(* Logix 5000 project; controller AplicacionAFEbancoDePruebas vendor 1 type 14 code 149 rev 33.12; software revision 33.01 *)

TASK MainTask (continuous, watchdog 500 ms) : MainProgram

MODULES
   Local : vendor 1 type 14 code 149 (Compact 0, rev 33.12)
      Discrete_IO : Embedded (Compact 1, rev 3.1, Output RPI 20 ms)
      PLC : 1769-L32E Ethernet Port (Ethernet 192.168.2.131, rev 20.1)
         PLC_Controller : vendor 1 type 14 code 77 (CompactLogixL32EController 0, rev 20.1, $6f3b489b$ RPI 20 ms, $fb73b292$ RPI 20 ms, $0a2ffb0d$ RPI 20 ms)
      VSD_AFE : vendor 1 type 143 code 8336 (Ethernet 192.168.2.50, rev 6.5, Output RPI 20 ms)
           VSD_AFE:O.LogicCommand_Stop   // Comando de Parada
           VSD_AFE:O.LogicCommand_Start   // Comando de Arranque
          : vendor 1 type 143 code 161 (RhinoBP 10, rev 1.1)
          : vendor 1 type 143 code 416 (RhinoBP 5, rev 1.8)
          : vendor 1 type 143 code 675 (RhinoBP 13, rev 1.1)
          : vendor 1 type 143 code 416 (RhinoBP 4, rev 1.8)
          : vendor 1 type 143 code 4770 (RhinoBP 12, rev 1.1)
          : vendor 1 type 143 code 2724 (RhinoBP 14, rev 1.1)
END_MODULES

TYPE Dinagrama :   // Estructura para el dinagrama
STRUCT
   vPotencia : REAL[500];   // captura del vector de potencia
   vCarga : REAL[500];   // captura del vector de carga
   vPosicion : REAL[500];   // captura del vector posicion
   vProximetro : DINT[500];   // captura del vector del proximetro
   NumeroMuestras : INT;
   enabled : BOOL;
   captura : BOOL;   // Flag que indica la captura del sistema
   resetVector : BOOL;   // Flag para darle Reset al vector de posición y carga
   vEmptyREAL : REAL[500];
   vEmptyINT : DINT[500];
   tMuestreo : REAL;   // Tiempo de Muestreo de captura
END_STRUCT
END_TYPE

TYPE LSW :   // Drive - Logic Status Word
STRUCT
   Faulted : BOOL;
   Warning : BOOL;
   RunForward : BOOL;
   RunReverse : BOOL;
   Ready : BOOL;
   RemoteRef : BOOL;
   RemoteCrtl : BOOL;
   AtSpeed : BOOL;
END_STRUCT
END_TYPE

TYPE SWC :
STRUCT
   Dinagrama : Dinagrama;
   VSD : VSD;
   entradasDigitales : INT;   // Entradas Digitales
   salidasDigitales : INT;   // Salidas Digitales
   entradasAnalogas : REAL[4];   // Entradas Analogas del PLC
   salidasAnalogas : REAL[4];
END_STRUCT
END_TYPE

TYPE VSD :   // VSD
STRUCT
   VSD_O : AB:PowerFlex755T_E_31635488:O:0;
   VSD_I : AB:PowerFlex755T_E_2B0A69C5:I:0;
END_STRUCT
END_TYPE

VAR_GLOBAL   (* controller tags *)
   SRP_Displacement_Actual : REAL := 22.99865;   // Variable de Simulacion PLC DC de Desplazamiento
   SRP_Load_Actual : REAL := 11.655421;   // Variable de simulacion PLC DC de Carga
   SRP_SimActualStroke : DINT;   // Variable Simulación de PLC Variador DC
   SWC : SWC := (Dinagrama.vCarga[0] := 9.6614, Dinagrama.vCarga[1] := 9.7812, Dinagrama.vCarga[2] := 9.711983, Dinagrama.vCarga[3] := 9.725293, Dinagrama.vCarga[4] := 9.842433, Dinagrama.vCarga[5] := 9.749254, Dinagrama.vCarga[6] := 9.69601, Dinagrama.vCarga[7] := 9.7306185, Dinagrama.vCarga[8] := 9.586858, Dinagrama.vCarga[9] := 9.751916, Dinagrama.vCarga[10] := 10.223133, Dinagrama.vCarga[11] := 10.473384, Dinagrama.vCarga[12] := 10.633119, Dinagrama.vCarga[13] := 10.856748, Dinagrama.vCarga[14] := 10.928628, Dinagrama.vCarga[15] := 11.109661, Dinagrama.vCarga[16] := 11.419147, Dinagrama.vCarga[17] := 11.515653, Dinagrama.vCarga[18] := 11.572558, Dinagrama.vCarga[19] := 11.751262, Dinagrama.vCarga[20] := 11.839782, Dinagrama.vCarga[21] := 11.974224, Dinagrama.vCarga[22] := 11.854091, Dinagrama.vCarga[23] := 11.607167, Dinagrama.vCarga[24] := 11.27239, Dinagrama.vCarga[25] := 11.069394, Dinagrama.vCarga[26] := 10.880708, Dinagrama.vCarga[27] := 10.662403, Dinagrama.vCarga[28] := 10.492021, Dinagrama.vCarga[29] := 10.321636, Dinagrama.vCarga[30] := 10.193849, Dinagrama.vCarga[31] := 10.018141, Dinagrama.vCarga[32] := 9.842432, Dinagrama.vCarga[33] := 9.682698, Dinagrama.vCarga[34] := 9.586857, Dinagrama.vCarga[35] := 9.706658, Dinagrama.vCarga[36] := 9.938273, Dinagrama.vCarga[37] := 10.113981, Dinagrama.vCarga[38] := 10.241769, Dinagrama.vCarga[39] := 10.321636, Dinagrama.vCarga[40] := 10.409491, Dinagrama.vCarga[41] := 10.409491, Dinagrama.vCarga[42] := 10.457411, Dinagrama.vCarga[43] := 10.534616, Dinagrama.vCarga[44] := 10.481371, Dinagrama.vCarga[45] := 10.555914, Dinagrama.vCarga[46] := 10.705, Dinagrama.vCarga[47] := 10.603834, Dinagrama.vCarga[48] := 10.316312, Dinagrama.vCarga[49] := 10.060737, Dinagrama.vCarga[50] := 9.970221, Dinagrama.vCarga[51] := 9.850419, Dinagrama.vCarga[52] := 9.608155, Dinagrama.vCarga[53] := 9.405825, Dinagrama.vCarga[54] := 9.389851, Dinagrama.vCarga[55] := 9.34193, Dinagrama.vCarga[56] := 9.131613, Dinagrama.vCarga[57] := 9.049084, Dinagrama.vCarga[58] := 9.08103, Dinagrama.vCarga[59] := 8.9266205,
        Dinagrama.vCarga[60] := 8.873376, Dinagrama.vCarga[61] := 9.155573, Dinagrama.vCarga[62] := 9.427122, Dinagrama.vCarga[63] := 9.549585, Dinagrama.vCarga[64] := 9.682697, Dinagrama.vCarga[65] := 9.906326, Dinagrama.vCarga[66] := 10.002167, Dinagrama.vCarga[67] := 9.980869, Dinagrama.vCarga[68] := 9.986194, Dinagrama.vCarga[69] := 9.980869, Dinagrama.vCarga[70] := 10.0208025, Dinagrama.vCarga[71] := 9.994181, Dinagrama.vCarga[72] := 10.098008, Dinagrama.vCarga[73] := 10.193849, Dinagrama.vCarga[74] := 9.938273, Dinagrama.vCarga[75] := 9.618804, Dinagrama.vCarga[76] := 9.538937, Dinagrama.vCarga[77] := 9.55491, Dinagrama.vCarga[78] := 9.331282, Dinagrama.vCarga[79] := 9.171547, Dinagrama.vCarga[80] := 9.347255, Dinagrama.vCarga[81] := 9.315308, Dinagrama.vCarga[82] := 9.123626, Dinagrama.vCarga[83] := 9.18752, Dinagrama.vCarga[84] := 9.331282, Dinagrama.vCarga[85] := 9.182196, Dinagrama.vCarga[86] := 9.166222, Dinagrama.vCarga[87] := 9.400499, Dinagrama.vCarga[88] := 9.693347, Dinagrama.vCarga[89] := 9.688023, Dinagrama.vCarga[90] := 9.746592, Dinagrama.vCarga[91] := 9.842432, Dinagrama.vCarga[92] := 9.885028, Dinagrama.vCarga[93] := 9.714644, Dinagrama.vCarga[94] := 9.634777, Dinagrama.vCarga[95] := 9.656075, Dinagrama.vCarga[96] := 9.496341, Dinagrama.vCarga[97] := 9.272713, Dinagrama.vCarga[98] := 9.128951, Dinagrama.vCarga[99] := 8.910647, Dinagrama.vCarga[100] := 8.434105, Dinagrama.vCarga[101] := 8.02412, Dinagrama.vCarga[102] := 7.936266, Dinagrama.vCarga[103] := 7.851074, Dinagrama.vCarga[104] := 7.5129685, Dinagrama.vCarga[105] := 7.302651, Dinagrama.vCarga[106] := 7.281353, Dinagrama.vCarga[107] := 7.238757, Dinagrama.vCarga[108] := 6.993831, Dinagrama.vCarga[109] := 6.706309, Dinagrama.vCarga[110] := 6.6796865, Dinagrama.vCarga[111] := 6.903315, Dinagrama.vCarga[112] := 7.1056457, Dinagrama.vCarga[113] := 7.3771944, Dinagrama.vCarga[114] := 7.773869, Dinagrama.vCarga[115] := 7.91763, Dinagrama.vCarga[116] := 7.909643, Dinagrama.vCarga[117] := 8.077365, Dinagrama.vCarga[118] := 8.300993, Dinagrama.vCarga[119] := 8.340926,
        Dinagrama.vCarga[120] := 8.460728, Dinagrama.vCarga[121] := 8.70033, Dinagrama.vCarga[122] := 8.79617, Dinagrama.vCarga[123] := 8.788184, Dinagrama.vCarga[124] := 8.77221, Dinagrama.vCarga[125] := 8.588515, Dinagrama.vCarga[126] := 8.38086, Dinagrama.vCarga[127] := 8.412807, Dinagrama.vCarga[128] := 8.420794, Dinagrama.vCarga[129] := 8.431443, Dinagrama.vCarga[130] := 8.476701, Dinagrama.vCarga[131] := 8.580528, Dinagrama.vCarga[132] := 8.497999, Dinagrama.vCarga[133] := 8.559231, Dinagrama.vCarga[134] := 8.591178, Dinagrama.vCarga[135] := 8.56988, Dinagrama.vCarga[136] := 8.631111, Dinagrama.vCarga[137] := 8.84409, Dinagrama.vCarga[138] := 9.081031, Dinagrama.vCarga[139] := 9.278037, Dinagrama.vCarga[140] := 9.325957, Dinagrama.vCarga[141] := 9.363229, Dinagrama.vCarga[142] := 9.618804, Dinagrama.vCarga[143] := 9.682698, Dinagrama.vCarga[144] := 9.682698, Dinagrama.vCarga[145] := 9.703996, Dinagrama.vCarga[146] := 9.703996, Dinagrama.vCarga[147] := 9.703996, Dinagrama.vCarga[148] := 9.703996, Dinagrama.vCarga[149] := 9.703996, Dinagrama.vCarga[150] := 9.703996, Dinagrama.vCarga[151] := 9.703996, Dinagrama.vCarga[152] := 9.703996, Dinagrama.vCarga[153] := 9.703996, Dinagrama.vCarga[154] := 9.703996, Dinagrama.vCarga[155] := 9.703996, Dinagrama.vCarga[156] := 9.703996, Dinagrama.vCarga[157] := 9.703996, Dinagrama.vCarga[158] := 9.703996, Dinagrama.vCarga[159] := 9.703996, Dinagrama.vCarga[160] := 9.703996, Dinagrama.vCarga[161] := 9.703996, Dinagrama.vCarga[162] := 9.703996, Dinagrama.vCarga[163] := 9.703996, Dinagrama.vCarga[164] := 9.703996, Dinagrama.vCarga[165] := 9.703996, Dinagrama.vCarga[166] := 9.703996, Dinagrama.vCarga[167] := 9.703996, Dinagrama.vCarga[168] := 9.703996, Dinagrama.vCarga[169] := 9.703996, Dinagrama.vCarga[170] := 9.703996, Dinagrama.vCarga[171] := 9.703996, Dinagrama.vCarga[172] := 9.703996, Dinagrama.vCarga[173] := 9.703996, Dinagrama.vCarga[174] := 9.703996, Dinagrama.vCarga[175] := 9.703996, Dinagrama.vCarga[176] := 9.703996, Dinagrama.vCarga[177] := 9.703996, Dinagrama.vCarga[178] := 9.703996, Dinagrama.vCarga[179] := 9.703996,
        Dinagrama.vCarga[180] := 9.703996, Dinagrama.vCarga[181] := 9.703996, Dinagrama.vCarga[182] := 9.703996, Dinagrama.vCarga[183] := 9.703996, Dinagrama.vCarga[184] := 9.703996, Dinagrama.vCarga[185] := 9.703996, Dinagrama.vCarga[186] := 9.703996, Dinagrama.vCarga[187] := 9.703996, Dinagrama.vCarga[188] := 9.703996, Dinagrama.vCarga[189] := 9.703996, Dinagrama.vCarga[190] := 9.703996, Dinagrama.vCarga[191] := 9.703996, Dinagrama.vCarga[192] := 9.703996, Dinagrama.vCarga[193] := 9.703996, Dinagrama.vCarga[194] := 9.703996, Dinagrama.vCarga[195] := 9.703996, Dinagrama.vCarga[196] := 9.703996, Dinagrama.vCarga[197] := 9.703996, Dinagrama.vCarga[198] := 9.703996, Dinagrama.vCarga[199] := 9.703996, Dinagrama.vCarga[200] := 9.703996, Dinagrama.vCarga[201] := 9.703996, Dinagrama.vCarga[202] := 9.703996, Dinagrama.vCarga[203] := 9.703996, Dinagrama.vCarga[204] := 9.703996, Dinagrama.vCarga[205] := 9.703996, Dinagrama.vCarga[206] := 9.703996, Dinagrama.vCarga[207] := 9.703996, Dinagrama.vCarga[208] := 9.703996, Dinagrama.vCarga[209] := 9.703996, Dinagrama.vCarga[210] := 9.703996, Dinagrama.vCarga[211] := 9.703996, Dinagrama.vCarga[212] := 9.703996, Dinagrama.vCarga[213] := 9.703996, Dinagrama.vCarga[214] := 9.703996, Dinagrama.vCarga[215] := 9.703996, Dinagrama.vCarga[216] := 9.703996, Dinagrama.vCarga[217] := 9.703996, Dinagrama.vCarga[218] := 9.703996, Dinagrama.vCarga[219] := 9.703996, Dinagrama.vCarga[220] := 9.703996, Dinagrama.vCarga[221] := 9.703996, Dinagrama.vCarga[222] := 9.703996, Dinagrama.vCarga[223] := 9.703996, Dinagrama.vCarga[224] := 9.703996, Dinagrama.vCarga[225] := 9.703996, Dinagrama.vCarga[226] := 9.703996, Dinagrama.vCarga[227] := 9.703996, Dinagrama.vCarga[228] := 9.703996, Dinagrama.vCarga[229] := 9.703996, Dinagrama.vCarga[230] := 9.703996, Dinagrama.vCarga[231] := 9.703996, Dinagrama.vCarga[232] := 9.703996, Dinagrama.vCarga[233] := 9.703996, Dinagrama.vCarga[234] := 9.703996, Dinagrama.vCarga[235] := 9.703996, Dinagrama.vCarga[236] := 9.703996, Dinagrama.vCarga[237] := 9.703996, Dinagrama.vCarga[238] := 9.703996, Dinagrama.vCarga[239] := 9.703996,
        Dinagrama.vCarga[240] := 9.703996, Dinagrama.vCarga[241] := 9.703996, Dinagrama.vCarga[242] := 9.703996, Dinagrama.vCarga[243] := 9.703996, Dinagrama.vCarga[244] := 9.703996, Dinagrama.vCarga[245] := 9.703996, Dinagrama.vCarga[246] := 9.703996, Dinagrama.vCarga[247] := 9.703996, Dinagrama.vCarga[248] := 9.703996, Dinagrama.vCarga[249] := 9.703996, Dinagrama.vCarga[250] := 9.703996, Dinagrama.vCarga[251] := 9.703996, Dinagrama.vCarga[252] := 9.703996, Dinagrama.vCarga[253] := 9.703996, Dinagrama.vCarga[254] := 9.703996, Dinagrama.vCarga[255] := 9.703996, Dinagrama.vCarga[256] := 9.703996, Dinagrama.vCarga[257] := 9.703996, Dinagrama.vCarga[258] := 9.703996, Dinagrama.vCarga[259] := 9.703996, Dinagrama.vCarga[260] := 9.703996, Dinagrama.vCarga[261] := 9.703996, Dinagrama.vCarga[262] := 9.703996, Dinagrama.vCarga[263] := 9.703996, Dinagrama.vCarga[264] := 9.703996, Dinagrama.vCarga[265] := 9.703996, Dinagrama.vCarga[266] := 9.703996, Dinagrama.vCarga[267] := 9.703996, Dinagrama.vCarga[268] := 9.703996, Dinagrama.vCarga[269] := 9.703996, Dinagrama.vCarga[270] := 9.703996, Dinagrama.vCarga[271] := 9.703996, Dinagrama.vCarga[272] := 9.703996, Dinagrama.vCarga[273] := 9.703996, Dinagrama.vCarga[274] := 9.703996, Dinagrama.vCarga[275] := 9.703996, Dinagrama.vCarga[276] := 9.703996, Dinagrama.vCarga[277] := 9.703996, Dinagrama.vCarga[278] := 9.703996, Dinagrama.vCarga[279] := 9.703996, Dinagrama.vCarga[280] := 9.703996, Dinagrama.vCarga[281] := 9.703996, Dinagrama.vCarga[282] := 9.703996, Dinagrama.vCarga[283] := 9.703996, Dinagrama.vCarga[284] := 9.703996, Dinagrama.vCarga[285] := 9.703996, Dinagrama.vCarga[286] := 9.703996, Dinagrama.vCarga[287] := 9.703996, Dinagrama.vCarga[288] := 9.703996, Dinagrama.vCarga[289] := 9.703996, Dinagrama.vCarga[290] := 9.703996, Dinagrama.vCarga[291] := 9.703996, Dinagrama.vPosicion[0] := 0.22007, Dinagrama.vPosicion[1] := 0.4084145, Dinagrama.vPosicion[2] := 0.8989175, Dinagrama.vPosicion[3] := 1.5143573, Dinagrama.vPosicion[4] := 2.2604218, Dinagrama.vPosicion[5] := 3.1391559, Dinagrama.vPosicion[6] := 4.147569, Dinagrama.vPosicion[7] := 5.2654533,
        Dinagrama.vPosicion[8] := 6.4805126, Dinagrama.vPosicion[9] := 7.78114, Dinagrama.vPosicion[10] := 9.158964, Dinagrama.vPosicion[11] := 10.613574, Dinagrama.vPosicion[12] := 12.155543, Dinagrama.vPosicion[13] := 13.778378, Dinagrama.vPosicion[14] := 14.611691, Dinagrama.vPosicion[15] := 16.600204, Dinagrama.vPosicion[16] := 19.2797, Dinagrama.vPosicion[17] := 21.118301, Dinagrama.vPosicion[18] := 22.049511, Dinagrama.vPosicion[19] := 23.956749, Dinagrama.vPosicion[20] := 25.906015, Dinagrama.vPosicion[21] := 27.897532, Dinagrama.vPosicion[22] := 29.92443, Dinagrama.vPosicion[23] := 32.000904, Dinagrama.vPosicion[24] := 34.121273, Dinagrama.vPosicion[25] := 36.271236, Dinagrama.vPosicion[26] := 38.454124, Dinagrama.vPosicion[27] := 40.67515, Dinagrama.vPosicion[28] := 42.926197, Dinagrama.vPosicion[29] := 45.59054, Dinagrama.vPosicion[30] := 47.925312, Dinagrama.vPosicion[31] := 50.300934, Dinagrama.vPosicion[32] := 52.57733, Dinagrama.vPosicion[33] := 54.853752, Dinagrama.vPosicion[34] := 57.161697, Dinagrama.vPosicion[35] := 58.29858, Dinagrama.vPosicion[36] := 60.54371, Dinagrama.vPosicion[37] := 63.858036, Dinagrama.vPosicion[38] := 66.06483, Dinagrama.vPosicion[39] := 67.1463, Dinagrama.vPosicion[40] := 69.277466, Dinagrama.vPosicion[41] := 71.36186, Dinagrama.vPosicion[42] := 73.41511, Dinagrama.vPosicion[43] := 75.75438, Dinagrama.vPosicion[44] := 77.68309, Dinagrama.vPosicion[45] := 79.54948, Dinagrama.vPosicion[46] := 81.36385, Dinagrama.vPosicion[47] := 83.1282, Dinagrama.vPosicion[48] := 84.8323, Dinagrama.vPosicion[49] := 86.45127, Dinagrama.vPosicion[50] := 87.23202, Dinagrama.vPosicion[51] := 88.73018, Dinagrama.vPosicion[52] := 90.154045, Dinagrama.vPosicion[53] := 92.103096, Dinagrama.vPosicion[54] := 93.29226, Dinagrama.vPosicion[55] := 93.858185, Dinagrama.vPosicion[56] := 94.9114, Dinagrama.vPosicion[57] := 96.00089, Dinagrama.vPosicion[58] := 96.84068, Dinagrama.vPosicion[59] := 97.581314, Dinagrama.vPosicion[60] := 98.21293, Dinagrama.vPosicion[61] := 98.7474, Dinagrama.vPosicion[62] := 99.18755, Dinagrama.vPosicion[63] := 99.53332, Dinagrama.vPosicion[64] := 99.77987, Dinagrama.vPosicion[65] := 99.935196, Dinagrama.vPosicion[66] := 99.983795, Dinagrama.vPosicion[67] := 99.96849,
        Dinagrama.vPosicion[68] := 99.8579, Dinagrama.vPosicion[69] := 99.64918, Dinagrama.vPosicion[70] := 99.51568, Dinagrama.vPosicion[71] := 99.1922, Dinagrama.vPosicion[72] := 98.72924, Dinagrama.vPosicion[73] := 98.26827, Dinagrama.vPosicion[74] := 97.74029, Dinagrama.vPosicion[75] := 97.14606, Dinagrama.vPosicion[76] := 96.499626, Dinagrama.vPosicion[77] := 95.795845, Dinagrama.vPosicion[78] := 95.004196, Dinagrama.vPosicion[79] := 94.16693, Dinagrama.vPosicion[80] := 93.305756, Dinagrama.vPosicion[81] := 92.36308, Dinagrama.vPosicion[82] := 91.377556, Dinagrama.vPosicion[83] := 90.37801, Dinagrama.vPosicion[84] := 89.32036, Dinagrama.vPosicion[85] := 88.01027, Dinagrama.vPosicion[86] := 87.43099, Dinagrama.vPosicion[87] := 86.2471, Dinagrama.vPosicion[88] := 85.00949, Dinagrama.vPosicion[89] := 83.06744, Dinagrama.vPosicion[90] := 81.722916, Dinagrama.vPosicion[91] := 81.02402, Dinagrama.vPosicion[92] := 79.59406, Dinagrama.vPosicion[93] := 78.12919, Dinagrama.vPosicion[94] := 76.61854, Dinagrama.vPosicion[95] := 75.04756, Dinagrama.vPosicion[96] := 73.44262, Dinagrama.vPosicion[97] := 71.8104, Dinagrama.vPosicion[98] := 70.117615, Dinagrama.vPosicion[99] := 68.385605, Dinagrama.vPosicion[100] := 66.349724, Dinagrama.vPosicion[101] := 64.541084, Dinagrama.vPosicion[102] := 63.614063, Dinagrama.vPosicion[103] := 61.744232, Dinagrama.vPosicion[104] := 58.907894, Dinagrama.vPosicion[105] := 56.94176, Dinagrama.vPosicion[106] := 55.949615, Dinagrama.vPosicion[107] := 53.960396, Dinagrama.vPosicion[108] := 51.950417, Dinagrama.vPosicion[109] := 49.88953, Dinagrama.vPosicion[110] := 47.795254, Dinagrama.vPosicion[111] := 45.690845, Dinagrama.vPosicion[112] := 43.56501, Dinagrama.vPosicion[113] := 42.49205, Dinagrama.vPosicion[114] := 38.891975, Dinagrama.vPosicion[115] := 36.722637, Dinagrama.vPosicion[116] := 34.528854, Dinagrama.vPosicion[117] := 32.329132, Dinagrama.vPosicion[118] := 30.155361, Dinagrama.vPosicion[119] := 27.987307, Dinagrama.vPosicion[120] := 25.821117, Dinagrama.vPosicion[121] := 23.68875, Dinagrama.vPosicion[122] := 21.607874, Dinagrama.vPosicion[123] := 19.584843, Dinagrama.vPosicion[124] := 17.632542, Dinagrama.vPosicion[125] := 15.761359, Dinagrama.vPosicion[126] := 13.965392, Dinagrama.vPosicion[127] := 12.251199,
        Dinagrama.vPosicion[128] := 10.367658, Dinagrama.vPosicion[129] := 8.857708, Dinagrama.vPosicion[130] := 8.136012, Dinagrama.vPosicion[131] := 6.7788615, Dinagrama.vPosicion[132] := 5.529149, Dinagrama.vPosicion[133] := 3.8806663, Dinagrama.vPosicion[134] := 3.3902075, Dinagrama.vPosicion[135] := 2.520764, Dinagrama.vPosicion[136] := 1.7710685, Dinagrama.vPosicion[137] := 1.148738, Dinagrama.vPosicion[138] := 0.66532767, Dinagrama.vPosicion[139] := 0.31461334, Dinagrama.vPosicion[140] := 0.096083336, Dinagrama.vPosicion[141] := 0.009929333, Dinagrama.vPosicion[142] := 0.049646668, Dinagrama.vPosicion[143] := 0.059576, Dinagrama.vPosicion[144] := 0.059576, Dinagrama.vPosicion[145] := 82.400505, Dinagrama.vPosicion[146] := 82.400505, Dinagrama.vPosicion[147] := 82.400505, Dinagrama.vPosicion[148] := 82.400505, Dinagrama.vPosicion[149] := 82.400505, Dinagrama.vPosicion[150] := 82.400505, Dinagrama.vPosicion[151] := 82.400505, Dinagrama.vPosicion[152] := 82.400505, Dinagrama.vPosicion[153] := 82.400505, Dinagrama.vPosicion[154] := 82.400505, Dinagrama.vPosicion[155] := 82.400505, Dinagrama.vPosicion[156] := 82.400505, Dinagrama.vPosicion[157] := 82.400505, Dinagrama.vPosicion[158] := 82.400505, Dinagrama.vPosicion[159] := 82.400505, Dinagrama.vPosicion[160] := 82.400505, Dinagrama.vPosicion[161] := 82.400505, Dinagrama.vPosicion[162] := 82.400505, Dinagrama.vPosicion[163] := 82.400505, Dinagrama.vPosicion[164] := 82.400505, Dinagrama.vPosicion[165] := 82.400505, Dinagrama.vPosicion[166] := 82.400505, Dinagrama.vPosicion[167] := 82.400505, Dinagrama.vPosicion[168] := 82.400505, Dinagrama.vPosicion[169] := 82.400505, Dinagrama.vPosicion[170] := 82.400505, Dinagrama.vPosicion[171] := 82.400505, Dinagrama.vPosicion[172] := 82.400505, Dinagrama.vPosicion[173] := 82.400505, Dinagrama.vPosicion[174] := 82.400505, Dinagrama.vPosicion[175] := 82.400505, Dinagrama.vPosicion[176] := 82.400505, Dinagrama.vPosicion[177] := 82.400505, Dinagrama.vPosicion[178] := 82.400505, Dinagrama.vPosicion[179] := 82.400505, Dinagrama.vPosicion[180] := 82.400505, Dinagrama.vPosicion[181] := 82.400505, Dinagrama.vPosicion[182] := 82.400505, Dinagrama.vPosicion[183] := 82.400505, Dinagrama.vPosicion[184] := 82.400505, Dinagrama.vPosicion[185] := 82.400505, Dinagrama.vPosicion[186] := 82.400505, Dinagrama.vPosicion[187] := 82.400505,
        Dinagrama.vPosicion[188] := 82.400505, Dinagrama.vPosicion[189] := 82.400505, Dinagrama.vPosicion[190] := 82.400505, Dinagrama.vPosicion[191] := 82.400505, Dinagrama.vPosicion[192] := 82.400505, Dinagrama.vPosicion[193] := 82.400505, Dinagrama.vPosicion[194] := 82.400505, Dinagrama.vPosicion[195] := 82.400505, Dinagrama.vPosicion[196] := 82.400505, Dinagrama.vPosicion[197] := 82.400505, Dinagrama.vPosicion[198] := 82.400505, Dinagrama.vPosicion[199] := 82.400505, Dinagrama.vPosicion[200] := 82.400505, Dinagrama.vPosicion[201] := 82.400505, Dinagrama.vPosicion[202] := 82.400505, Dinagrama.vPosicion[203] := 82.400505, Dinagrama.vPosicion[204] := 82.400505, Dinagrama.vPosicion[205] := 82.400505, Dinagrama.vPosicion[206] := 82.400505, Dinagrama.vPosicion[207] := 82.400505, Dinagrama.vPosicion[208] := 82.400505, Dinagrama.vPosicion[209] := 82.400505, Dinagrama.vPosicion[210] := 82.400505, Dinagrama.vPosicion[211] := 82.400505, Dinagrama.vPosicion[212] := 82.400505, Dinagrama.vPosicion[213] := 82.400505, Dinagrama.vPosicion[214] := 82.400505, Dinagrama.vPosicion[215] := 82.400505, Dinagrama.vPosicion[216] := 82.400505, Dinagrama.vPosicion[217] := 82.400505, Dinagrama.vPosicion[218] := 82.400505, Dinagrama.vPosicion[219] := 82.400505, Dinagrama.vPosicion[220] := 82.400505, Dinagrama.vPosicion[221] := 82.400505, Dinagrama.vPosicion[222] := 82.400505, Dinagrama.vPosicion[223] := 82.400505, Dinagrama.vPosicion[224] := 82.400505, Dinagrama.vPosicion[225] := 82.400505, Dinagrama.vPosicion[226] := 82.400505, Dinagrama.vPosicion[227] := 82.400505, Dinagrama.vPosicion[228] := 82.400505, Dinagrama.vPosicion[229] := 82.400505, Dinagrama.vPosicion[230] := 82.400505, Dinagrama.vPosicion[231] := 82.400505, Dinagrama.vPosicion[232] := 82.400505, Dinagrama.vPosicion[233] := 82.400505, Dinagrama.vPosicion[234] := 82.400505, Dinagrama.vPosicion[235] := 82.400505, Dinagrama.vPosicion[236] := 82.400505, Dinagrama.vPosicion[237] := 82.400505, Dinagrama.vPosicion[238] := 82.400505, Dinagrama.vPosicion[239] := 82.400505, Dinagrama.vPosicion[240] := 82.400505, Dinagrama.vPosicion[241] := 82.400505, Dinagrama.vPosicion[242] := 82.400505, Dinagrama.vPosicion[243] := 82.400505, Dinagrama.vPosicion[244] := 82.400505, Dinagrama.vPosicion[245] := 82.400505, Dinagrama.vPosicion[246] := 82.400505, Dinagrama.vPosicion[247] := 82.400505,
        Dinagrama.vPosicion[248] := 82.400505, Dinagrama.vPosicion[249] := 82.400505, Dinagrama.vPosicion[250] := 82.400505, Dinagrama.vPosicion[251] := 82.400505, Dinagrama.vPosicion[252] := 82.400505, Dinagrama.vPosicion[253] := 82.400505, Dinagrama.vPosicion[254] := 82.400505, Dinagrama.vPosicion[255] := 82.400505, Dinagrama.vPosicion[256] := 82.400505, Dinagrama.vPosicion[257] := 82.400505, Dinagrama.vPosicion[258] := 82.400505, Dinagrama.vPosicion[259] := 82.400505, Dinagrama.vPosicion[260] := 82.400505, Dinagrama.vPosicion[261] := 82.400505, Dinagrama.vPosicion[262] := 82.400505, Dinagrama.vPosicion[263] := 82.400505, Dinagrama.vPosicion[264] := 82.400505, Dinagrama.vPosicion[265] := 82.400505, Dinagrama.vPosicion[266] := 82.400505, Dinagrama.vPosicion[267] := 82.400505, Dinagrama.vPosicion[268] := 82.400505, Dinagrama.vPosicion[269] := 82.400505, Dinagrama.vPosicion[270] := 82.400505, Dinagrama.vPosicion[271] := 82.400505, Dinagrama.vPosicion[272] := 82.400505, Dinagrama.vPosicion[273] := 82.400505, Dinagrama.vPosicion[274] := 82.400505, Dinagrama.vPosicion[275] := 82.400505, Dinagrama.vPosicion[276] := 82.400505, Dinagrama.vPosicion[277] := 82.400505, Dinagrama.vPosicion[278] := 82.400505, Dinagrama.vPosicion[279] := 82.400505, Dinagrama.vPosicion[280] := 82.400505, Dinagrama.vPosicion[281] := 82.400505, Dinagrama.vPosicion[282] := 82.400505, Dinagrama.vPosicion[283] := 82.400505, Dinagrama.vPosicion[284] := 82.400505, Dinagrama.vPosicion[285] := 82.400505, Dinagrama.vPosicion[286] := 82.400505, Dinagrama.vPosicion[287] := 82.400505, Dinagrama.vPosicion[288] := 82.400505, Dinagrama.vPosicion[289] := 82.400505, Dinagrama.vPosicion[290] := 82.400505, Dinagrama.vPosicion[291] := 82.400505, Dinagrama.vProximetro[0] := 1, Dinagrama.vProximetro[1] := 1, Dinagrama.vProximetro[2] := 1, Dinagrama.vProximetro[143] := 1, Dinagrama.NumeroMuestras := 143, Dinagrama.enabled := 1, Dinagrama.tMuestreo := 0.05, VSD.VSD_O.P10_VRefAStpt := 59.4079, VSD.VSD_I.DriveStatus := 2#0010_0001_0000_0000_0000_0100_0000_1101, VSD.VSD_I.DriveStatus_Ready := 1, VSD.VSD_I.DriveStatus_CommandDir := 1, VSD.VSD_I.DriveStatus_ActualDir := 1, VSD.VSD_I.DriveStatus_SpdRefBit0 := 1, VSD.VSD_I.DriveStatus_AtZeroSpeed := 1, VSD.VSD_I.DriveStatus_EnableOn := 1, VSD.VSD_I.P10_VRefCommanded := 59.407898,
        VSD.VSD_I.DCBusVolts := 700.00836, VSD.VSD_I.P10_HeatsnkTemp := 22.376202, VSD.VSD_I.ElapsedRunTime := 29.436, VSD.VSD_I.LastFaultCode := 13065, VSD.VSD_I.ElapsedkWH := -20501, entradasDigitales := 3, entradasAnalogas[0] := -1.7e-44, entradasAnalogas[1] := -9.176336e+29, entradasAnalogas[2] := 3.8693e-41, entradasAnalogas[3] := 6.66079e-40, salidasAnalogas[0] := 1.e-45, salidasAnalogas[1] := 6.e-45, salidasAnalogas[2] := 4.e-45);
        .Dinagrama.enabled   // Habilitar Adquision
END_VAR

PROGRAM MainProgram   (* main routine R000_MainRoutine *)
VAR
   Captura : BOOL;
   contadorAux : ALIAS FOR counter[0].ACC;
   counter : COUNTER[10];
   Enabled : BOOL;
   Flag : BOOL;
   habilitar : DINT;
   myoneshot : BOOL[32] := ([1] := 1, [2] := 1);
        [0]   // oneshot toogle bot dinagrama
        [1]   // oneshor reset del ocntador
        [2]   // reset de la flag cuando se habilita y se deshabilita
   Proximetro_Virtual : ALIAS FOR SRP_SimActualStroke;
   SPM_Reference : REAL := 8.5;
   timer : TIMER[10] := ([0].PRE := 50);
        [0]   // Tiempo Muestreo
END_VAR

ROUTINE R000_MainRoutine   (* ladder *)
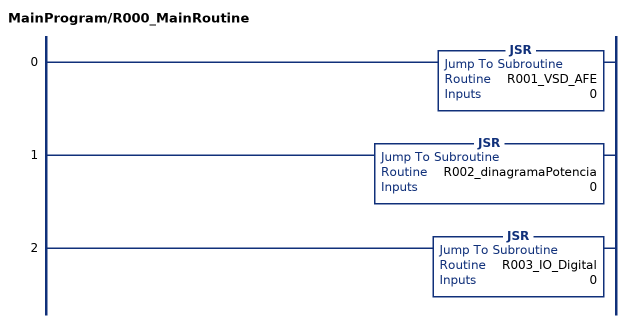
   0: JSR(R001_VSD_AFE,0);
   1: JSR(R002_dinagramaPotencia,0);
   2: JSR(R003_IO_Digital,0);
END_ROUTINE

ROUTINE R001_VSD_AFE   (* ladder *)
// Comandos Basicos de Operación de VSD AFE
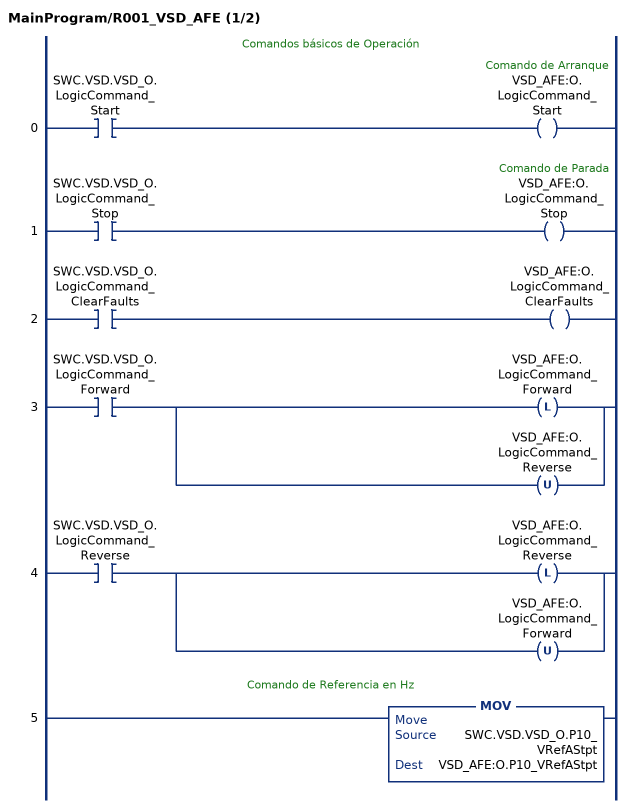
   // Comandos básicos de Operación
   0: XIC(SWC.VSD.VSD_O.LogicCommand_Start)OTE(VSD_AFE:O.LogicCommand_Start);
   1: XIC(SWC.VSD.VSD_O.LogicCommand_Stop)OTE(VSD_AFE:O.LogicCommand_Stop);
   2: XIC(SWC.VSD.VSD_O.LogicCommand_ClearFaults)OTE(VSD_AFE:O.LogicCommand_ClearFaults);
   3: XIC(SWC.VSD.VSD_O.LogicCommand_Forward)[OTL(VSD_AFE:O.LogicCommand_Forward) ,OTU(VSD_AFE:O.LogicCommand_Reverse) ];
   4: XIC(SWC.VSD.VSD_O.LogicCommand_Reverse)[OTL(VSD_AFE:O.LogicCommand_Reverse) ,OTU(VSD_AFE:O.LogicCommand_Forward) ];
   // Comando de Referencia en Hz
   5: MOV(SWC.VSD.VSD_O.P10_VRefAStpt,VSD_AFE:O.P10_VRefAStpt);
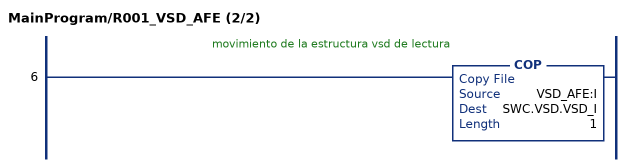
   // movimiento de la estructura vsd de lectura
   6: COP(VSD_AFE:I,SWC.VSD.VSD_I,1);
END_ROUTINE

ROUTINE R002_dinagramaPotencia   (* ladder *)
// Adquisión de los diferentes strokes para la captura del dinagrama de superficie
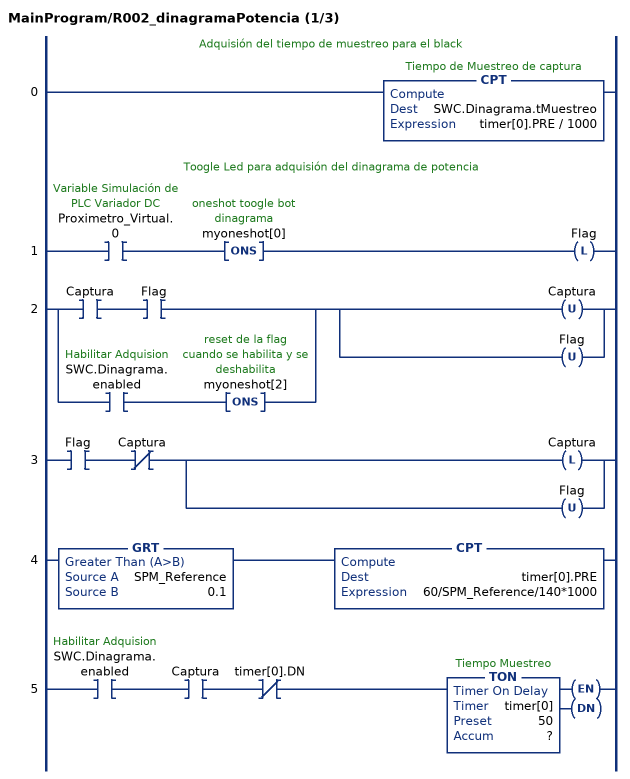
   // Adquisión del tiempo de muestreo para el black
   0: CPT(SWC.Dinagrama.tMuestreo,timer[0].PRE / 1000);
   // Toogle Led para adquisión del dinagrama de potencia
   1: XIC(Proximetro_Virtual.0)ONS(myoneshot[0])OTL(Flag);
   2: [XIC(Captura) XIC(Flag) ,XIC(SWC.Dinagrama.enabled) ONS(myoneshot[2]) ][OTU(Captura) ,OTU(Flag) ];
   3: XIC(Flag)XIO(Captura)[OTL(Captura) ,OTU(Flag) ];
   4: GRT(SPM_Reference,0.1)CPT(timer[0].PRE,60/SPM_Reference/140*1000);
   5: XIC(SWC.Dinagrama.enabled)XIC(Captura)XIO(timer[0].DN)TON(timer[0],?,?);
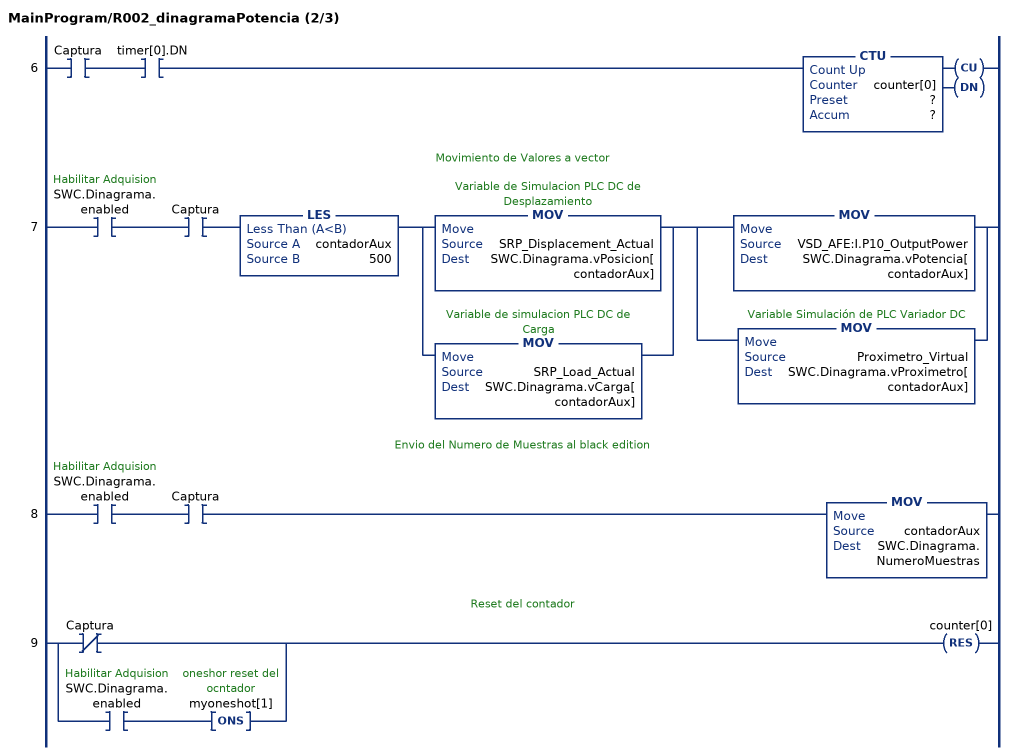
   6: XIC(Captura)XIC(timer[0].DN)CTU(counter[0],?,?);
   // Movimiento de Valores a vector
   7: XIC(SWC.Dinagrama.enabled)XIC(Captura)LES(contadorAux,500)[MOV(SRP_Displacement_Actual,SWC.Dinagrama.vPosicion[contadorAux]) ,MOV(SRP_Load_Actual,SWC.Dinagrama.vCarga[contadorAux]) ][MOV(VSD_AFE:I.P10_OutputPower,SWC.Dinagrama.vPotencia[contadorAux]) ,MOV(Proximetro_Virtual,SWC.Dinagrama.vProximetro[contadorAux]) ];
   // Envio del Numero de Muestras al black edition
   8: XIC(SWC.Dinagrama.enabled)XIC(Captura)MOV(contadorAux,SWC.Dinagrama.NumeroMuestras);
   // Reset del contador
   9: [XIO(Captura) ,XIC(SWC.Dinagrama.enabled) ONS(myoneshot[1]) ]RES(counter[0]);
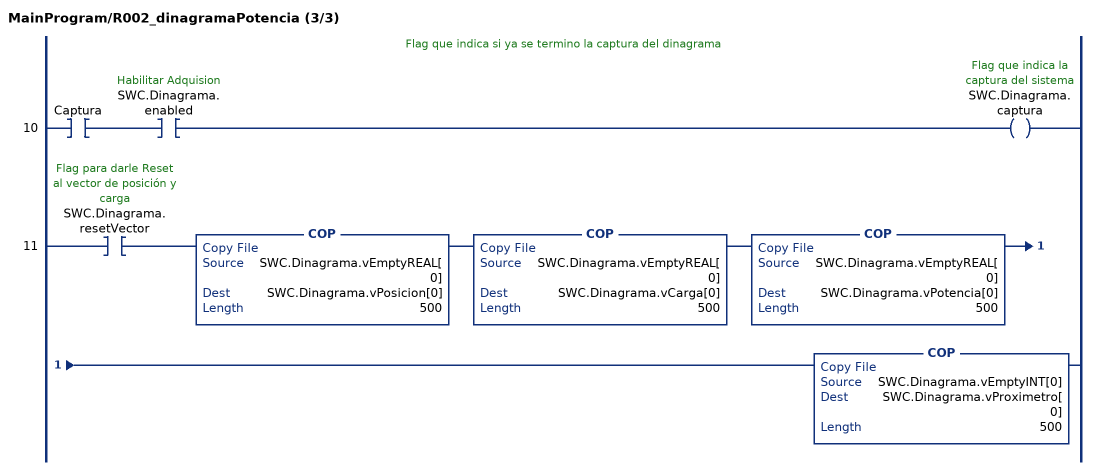
   // Flag que indica si ya se termino la captura del dinagrama
   10: XIC(Captura)XIC(SWC.Dinagrama.enabled)OTE(SWC.Dinagrama.captura);
   11: XIC(SWC.Dinagrama.resetVector)COP(SWC.Dinagrama.vEmptyREAL[0],SWC.Dinagrama.vPosicion[0],500)COP(SWC.Dinagrama.vEmptyREAL[0],SWC.Dinagrama.vCarga[0],500)COP(SWC.Dinagrama.vEmptyREAL[0],SWC.Dinagrama.vPotencia[0],500)COP(SWC.Dinagrama.vEmptyINT[0],SWC.Dinagrama.vProximetro[0],500);
END_ROUTINE

ROUTINE R003_IO_Digital   (* ladder *)
// Entradas Digitales
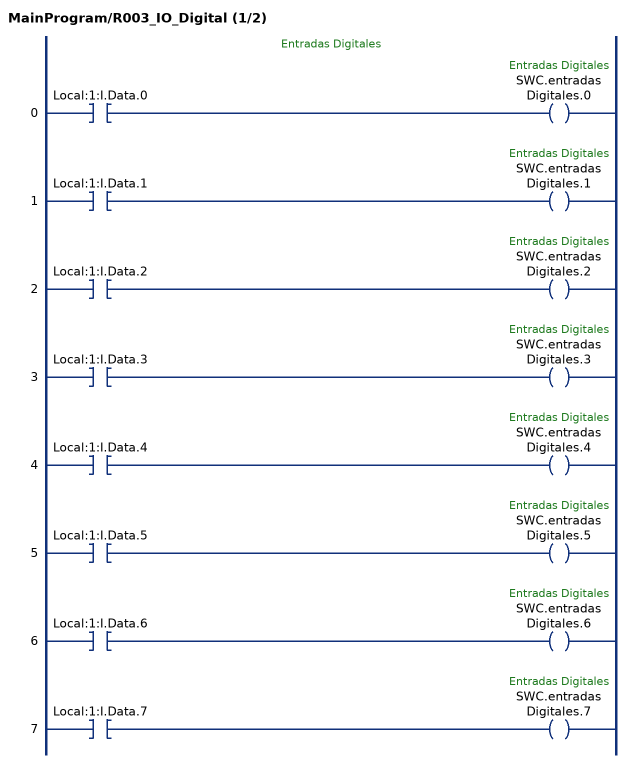
   // Entradas Digitales
   0: XIC(Local:1:I.Data.0)OTE(SWC.entradasDigitales.0);
   1: XIC(Local:1:I.Data.1)OTE(SWC.entradasDigitales.1);
   2: XIC(Local:1:I.Data.2)OTE(SWC.entradasDigitales.2);
   3: XIC(Local:1:I.Data.3)OTE(SWC.entradasDigitales.3);
   4: XIC(Local:1:I.Data.4)OTE(SWC.entradasDigitales.4);
   5: XIC(Local:1:I.Data.5)OTE(SWC.entradasDigitales.5);
   6: XIC(Local:1:I.Data.6)OTE(SWC.entradasDigitales.6);
   7: XIC(Local:1:I.Data.7)OTE(SWC.entradasDigitales.7);
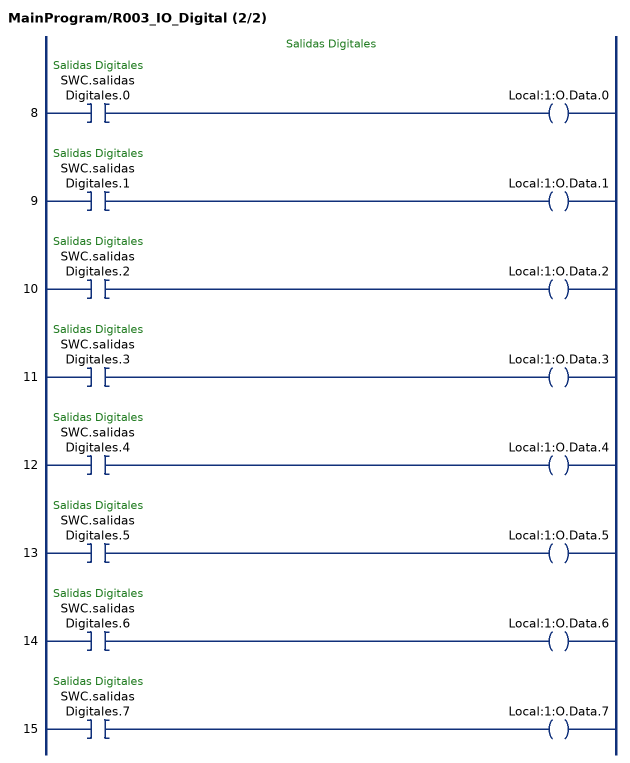
   // Salidas Digitales
   8: XIC(SWC.salidasDigitales.0)OTE(Local:1:O.Data.0);
   9: XIC(SWC.salidasDigitales.1)OTE(Local:1:O.Data.1);
   10: XIC(SWC.salidasDigitales.2)OTE(Local:1:O.Data.2);
   11: XIC(SWC.salidasDigitales.3)OTE(Local:1:O.Data.3);
   12: XIC(SWC.salidasDigitales.4)OTE(Local:1:O.Data.4);
   13: XIC(SWC.salidasDigitales.5)OTE(Local:1:O.Data.5);
   14: XIC(SWC.salidasDigitales.6)OTE(Local:1:O.Data.6);
   15: XIC(SWC.salidasDigitales.7)OTE(Local:1:O.Data.7);
END_ROUTINE
END_PROGRAM
